{attribute 'pack_mode' := '1'} 
TYPE ASCF_CC_OPCUACS_Reader_Temp_Dint :
STRUCT
	stReadListReturnInfo	: ARRAY [1..2] OF ST_UAReadListReturnInfo;
	QC		: BYTE	:= 16#0;
	Value	: DINT	:= 0;
END_STRUCT
END_TYPE

(* stored: Version 1.1.0.1, ProductVersion 3.1.4026.4
   DUT ASCF_CC_OPCUACS_Reader_Temp_Dint: Id {0ae3cb01-0f0b-4d87-8abc-1ebfd9041a04} *)
